SUBAPPLICATION Uebung_083 (* Beispiel für E_CTUD_UDINT *)
  (* Standard: 61499-2; Description: Copyright (c) 2023 Meisterschulen am Ostbahnhof This program and the accompanying materials are made available under the terms of the Eclipse Public License 2.0 which is available at https://www.eclipse.org/legal/epl-2.0/ SPDX-License-Identifier: EPL-2.0 Beispiel für E_CTD Aufwärts zählen UAO Curriculum Module 3 - The IEC 61499 Standard, Seite 94 *)
  (* Version 1.0, 2023-10-23, Franz Höpfinger, Meisterschulen am Ostbahnhof *)
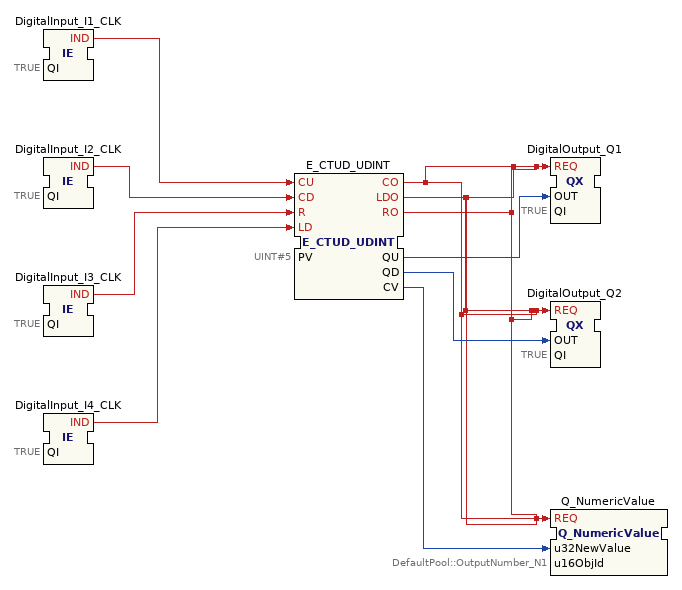
  FBS
    DigitalOutput_Q1 : QX(QI := TRUE);
    DigitalInput_I1_CLK : IE(QI := TRUE);
    E_CTUD_UDINT : E_CTUD_UDINT(PV := UINT#5);
    DigitalInput_I2_CLK : IE(QI := TRUE);
    DigitalInput_I3_CLK : IE(QI := TRUE);
    DigitalInput_I4_CLK : IE(QI := TRUE);
    DigitalOutput_Q2 : QX(QI := TRUE);
    Q_NumericValue : Q_NumericValue(u16ObjId := DefaultPool::OutputNumber_N1);
  END_FBS
  EVENT_CONNECTIONS
    DigitalInput_I1_CLK.IND TO E_CTUD_UDINT.CU;
    E_CTUD_UDINT.CO TO DigitalOutput_Q1.REQ;
    E_CTUD_UDINT.LDO TO DigitalOutput_Q1.REQ;
    DigitalInput_I2_CLK.IND TO E_CTUD_UDINT.CD;
    E_CTUD_UDINT.RO TO DigitalOutput_Q1.REQ;
    DigitalInput_I3_CLK.IND TO E_CTUD_UDINT.R;
    DigitalInput_I4_CLK.IND TO E_CTUD_UDINT.LD;
    E_CTUD_UDINT.LDO TO DigitalOutput_Q2.REQ;
    E_CTUD_UDINT.CO TO DigitalOutput_Q2.REQ;
    E_CTUD_UDINT.RO TO DigitalOutput_Q2.REQ;
    E_CTUD_UDINT.CO TO Q_NumericValue.REQ;
    E_CTUD_UDINT.RO TO Q_NumericValue.REQ;
    E_CTUD_UDINT.LDO TO Q_NumericValue.REQ;
  END_CONNECTIONS
  DATA_CONNECTIONS
    E_CTUD_UDINT.QU TO DigitalOutput_Q1.OUT;
    E_CTUD_UDINT.QD TO DigitalOutput_Q2.OUT;
    E_CTUD_UDINT.CV TO Q_NumericValue.u32NewValue;
  END_CONNECTIONS
END_SUBAPPLICATION
